{attribute addProperty BoxType "EL3632-0000-0016"}
{attribute addProperty Id "Ch1_Sample_CountAT %I*UINT162"}
{attribute addProperty CRC "2141697771"}
{attribute addProperty SizeInBites "16"}
{attribute addProperty SizeInBytes "2"}
TYPE Sample_Count_7FA7B6EB :
STRUCT
	{attribute addProperty Name "Ch1_Sample_Count"}
	Ch1_Sample_Count AT %I* : UINT;
END_STRUCT
END_TYPE

(* stored: Version 1.2.0.0, ProductVersion 3.1.4024.9
   DUT Sample_Count_7FA7B6EB: Id {89cbf72f-e181-4a91-86a5-a235067c4644} *)
